FUNCTION_BLOCK VesselControlFB
VAR_INPUT	
END_VAR
VAR_OUTPUT	
END_VAR
VAR			
iPressureLimitVessel_2_Min : INT; 		//Temp Variables for Vessel2 Pressure Control 
iPressureLimitVessel_2_Max : INT; 		//Temp Variables for Vessel2 Pressure Control 	
AutoManPushButton_rTrig : R_TRIG ;			//Button Rise Edge Read
END_VAR
VAR CONSTANT 
cAutoLimitMinPressureVessel2 : INT :=40; // Automatic Pressure Control Constant MIN
cAutoLimitMaxPressureVessel2 : INT :=60; // Automatic Pressure Control Constant MAX
cOneBar : INT :=1;						// Constant 1 Bar 
iAutoMode : INT := 1;
iManualMode : INT := 0;
END_VAR

//=============================================================================
// Dmitri Raihtsaum - Copyright 2023
// Created By: Dmitri Raihtsaum
//-----------------------------------------------------------------------------
// Tested with:   Twincat3, UaExpert
// Engineering:   Twincat3
// Functionality: Test Home Work - Vessel Pressure Control
// Date: 20.07.2023
// Rev 0.1
//=============================================================================

AutoManPushButton_rTrig(CLK :=  gOpc.Buttons.ModeButton); 		//Button Rise Edge Read
// System Mode Control
// push button for toggling the state between AUTOMATIC and MANUAL.
IF AutoManPushButton_rTrig.Q AND gopc.SystemState = iAutoMode THEN  			//Change From Auto To Manual
	gopc.SystemState := iManualMode;											//Change From Auto To Manual
ELSIF AutoManPushButton_rTrig.Q AND gopc.SystemState = iManualMode THEN		//Change From Manual To Auto
	gopc.SystemState:= iAutoMode; 											//Change From Manual To Auto
END_IF;
//Vessel 1 Control
// The pressure must be equal in both vessels ± 1 bar.
// Pressure in Vessel 1 is controlled in reference to Vessel 2 pressure:
// When pressure in Vessel 1 is 1 bar higher than is Vessel 2, then the Vessel 1
//valve shall be opened to release the pressure until the pressure in Vessel 1
//in 1 bar lower than the pressure in Vessel 2.

IF gOpc.Vessel[1].In.Sensor  >=  gOpc.Vessel[2].In.Sensor + cOneBar  THEN // Pressure Comparation Vessel1 and Vessel2 
	gOpc.Vessel[1].Out.Valves  :=TRUE;									  //Open Valve Y1
END_IF;

IF gOpc.Vessel[1].In.Sensor  <=  gOpc.Vessel[2].In.Sensor - cOneBar  THEN // Pressure Comparation Vessel1 and Vessel2
	gOpc.Vessel[1].Out.Valves  := FALSE;								  //Close Valve Y1
END_IF;
//Vessel 2 Control
//• Pressure in Vessel 2 is controlled in REFERENCE TO MIN AND MAX pressure
//parameters:
//o When pressure in Vessel 2 reaches Max parameter, then the Vessel 2 valve
//shall be opened to release the pressure until the pressure in Vessel 2
//reaches Min parameter.
//• The system shall have 2 states:
//o AUTOMATIC Min and Max parameters for Vessel 2 are given as
//constants 40 bar and 60 bar correspondingly.
//o MANUAL Min and Max parameters for Vessel 2 are given by Button 1
//(analogue potentiometer knob) and Button 2 (analogue potentiometer
//knob).
//o The state shall be changed using a third button (push button).
IF gopc.SystemState= iManualMode THEN 
	iPressureLimitVessel_2_Min := gOpc.Buttons.AnalogButtons[1];   //Temp Varibles data sellection
	iPressureLimitVessel_2_Max := gOpc.Buttons.AnalogButtons[2];	//Temp Varibles data sellection
END_IF;
IF gopc.SystemState = iAutoMode THEN 
	iPressureLimitVessel_2_Min := cAutoLimitMinPressureVessel2;			//Temp Varibles data sellection
	iPressureLimitVessel_2_Max := cAutoLimitMaxPressureVessel2;			//Temp Varibles data sellection
END_IF;
IF gOpc.Vessel[2].In.Sensor  >= iPressureLimitVessel_2_Max THEN  // Pressure Comparation  Vessel2 and Limits
	gOpc.Vessel[2].Out.Valves  :=TRUE;												//Open Valve Y2
END_IF
IF gOpc.Vessel[2].In.Sensor <= iPressureLimitVessel_2_MIN THEN // Pressure Comparation  Vessel2 and Limits
	gOpc.Vessel[2].Out.Valves  :=FALSE;											//Close Valve Y2
END_IF

//=============================================================================
//END
//=============================================================================

END_FUNCTION_BLOCK

(* stored: Version 1.1.0.1, ProductVersion 3.1.4024.12
   POU VesselControlFB: Id {e6bb8feb-d04d-47cd-95d4-09d5ffa70f50}, SpecialFunc None *)
